(* IEC 61131-3 sources: programs/VI-54/VI-54_20171205/VI-54_20171205/Stations/PLC_VI54/VI-54_171014/Class/Banner_EZlight, 1 file *)

(* ---- Banner_EZlight.st ---- *)
(*!
<Class
	Name               = "Banner_EZlight"
	Revision           = "0.0"
	RealtimeTask       = "false"
	CyclicTask         = "false"
	BackgroundTask     = "false"
	Sigmatek           = "false"
	OSInterface        = "false"
	HighPriority       = "false"
	Automatic          = "false"
	UpdateMode         = "Prescan"
	SharedCommandTable = "true"
	Objectsize         = "(480,120)">
	<Channels>
		<Server Name="ClassSvr" Visualized="false" Initialize="false" WriteProtected="true" Retentive="false"/>
		<Client Name="oCollorBlue" Required="false" Internal="false"/>
		<Client Name="oCollorGreen" Required="false" Internal="false"/>
		<Client Name="oCollorRed" Required="false" Internal="false"/>
		<Client Name="oCollorWhite" Required="false" Internal="false"/>
		<Client Name="oCollorYellow" Required="false" Internal="false"/>
	</Channels>
</Class>
*)
Banner_EZlight : CLASS
	TYPE
	  eLightCollor :  //! <Type Public="true" Name="eLightCollor"/>
	  (
	    eGreenOn,
	    eGreenFlashing,
	    eRedOn,
	    eRedFlashing,
	    eYellowOn,
	    eYellowFlashing,
	    eBlueOn,
	    eBlueFlashing,
	    eWhiteOn,
	    eWhiteFlashing,
	    eGreenRedFlashCycle,
	    eGreenYellowFlashCycle,
	    eGreenBlueFlashCycle,
	    eGreenWhiteFlashCycle,
	    eRedYellowFlashCycle,
	    eRedBlueFlashCycle,
	    eRedWhiteFlashCylce,
	    eYellowBlueFlashCycle,
	    eYellowWhiteFlashCycle,
	    eBlueWhiteFlashCycle
	  )$UDINT;
	END_TYPE
  //Servers:
	ClassSvr 	: SvrChCmd_DINT;
  //Clients:
	oCollorGreen 	: CltCh_DINT;
	oCollorRed 	: CltCh_DINT;
	oCollorYellow 	: CltCh_DINT;
	oCollorBlue 	: CltCh_DINT;
	oCollorWhite 	: CltCh_DINT;
  //Variables:
		State 	: eLightCollor;
		Oldstate 	: eLightCollor;
		GreenCollor 	: DINT;
		RedCollor 	: DINT;
		YellowCollor 	: DINT;
		BlueCollor 	: DINT;
		WhiteCollor 	: DINT;
  //Functions:

	FUNCTION VIRTUAL GLOBAL Init;

	FUNCTION GLOBAL LightCollors
		VAR_INPUT
			iCollor 	: eLightCollor;
		END_VAR;
  //Tables:
	FUNCTION @STD
		VAR_OUTPUT
			ret_code	: CONFSTATES;
		END_VAR;
	FUNCTION GLOBAL TAB @CT_;
END_CLASS;

FUNCTION VIRTUAL GLOBAL Banner_EZlight::Init

  // When starting up, give undefind value
  OldState$dint := -1;

END_FUNCTION

FUNCTION GLOBAL Banner_EZlight::LightCollors
	VAR_INPUT
		iCollor 	: eLightCollor;
	END_VAR

  // if state is different
  State := iCollor;
  if OldState <> State then
    Oldstate := State;

    // Set everything to zero
    GreenCollor   := 0;
    RedCollor     := 0;
    YellowCollor  := 0;
    BlueCollor    := 0;
    WhiteCollor   := 0;
  end_if;

  case State of
    eGreenOn:
      GreenCollor   := 1;

    eGreenFlashing:
      GreenCollor   := 1;
      RedCollor     := 1;

    eRedOn:
      RedCollor     := 1;

    eRedFlashing:
      RedCollor     := 1;
      YellowCollor  := 1;

    eYellowOn:
      YellowCollor  := 1;

    eYellowFlashing:
      YellowCollor  := 1;
      BlueCollor    := 1;

    eBlueOn:
      BlueCollor    := 1;

    eBlueFlashing:
      BlueCollor    := 1;
      WhiteCollor   := 1;

    eWhiteOn:
      WhiteCollor   := 1;

    eWhiteFlashing:
      WhiteCollor   := 1;
      GreenCollor   := 1;

    eGreenRedFlashCycle:
      GreenCollor   := 1;
      YellowCollor  := 1;

    eGreenYellowFlashCycle:
      GreenCollor   := 1;
      BlueCollor    := 1;

    eGreenBlueFlashCycle:
      RedCollor     := 1;
      BlueCollor    := 1;

    eGreenWhiteFlashCycle:
      RedCollor     := 1;
      WhiteCollor   := 1;

    eRedYellowFlashCycle:
      YellowCollor  := 1;
      WhiteCollor   := 1;

    eRedBlueFlashCycle:
      GreenCollor   := 1;
      RedCollor     := 1;
      WhiteCollor   := 1;

    eRedWhiteFlashCylce:
      GreenCollor   := 1;
      RedCollor     := 1;
      BlueCollor    := 1;

    eYellowBlueFlashCycle:
      GreenCollor   := 1;
      RedCollor     := 1;
      YellowCollor  := 1;

    eYellowWhiteFlashCycle:
      RedCollor     := 1;
      YellowCollor  := 1;
      WhiteCollor   := 1;

    eBlueWhiteFlashCycle:
      RedCollor     := 1;
      YellowCollor  := 1;
      WhiteCollor   := 1;
  end_case;

  // Set outputs
  oCollorGreen.Write(input:= GreenCollor);
  oCollorRed.Write(input:= RedCollor);
  oCollorYellow.Write(input:= YellowCollor);
  oCollorBlue.Write(input:= BlueCollor);
  oCollorWhite.Write(input:= WhiteCollor);

END_FUNCTION
